// TIA Portal V17 export
// export: Created 2023-04-07T09:30:35.0113751Z, ExportSetting WithDefaults, DisplayName Totally Integrated Automation Portal, DisplayVersion V17 Update 4, DisplayName TIA Portal Openness, DisplayVersion V17 Update 4, DisplayName TIA Portal Version Control Interface, DisplayVersion V17, DisplayName STEP 7 Professional, DisplayVersion V17 Update 4, DisplayName STEP 7 Safety, DisplayVersion V17, DisplayName WinCC Professional, DisplayVersion V17 Update 4
TYPE "W_PE"
// stored: IsFailsafeCompliant false
   STRUCT
      iUserPswIns : Int;   // To check / 40005
      iModePctrlCmd : Int := 0;   // Register 40861 / 40551
      iModeQctrlCmd : Int := 0;   // Register 40862 / 40552
      rPacRef : Real := 0.0;   // Register 40863 / 40553
      rQacRef : Real := 0.0;   // Register 40864 / 40558
      xStartCmd : Bool;   // Register 40040
      xGeneral_SelectorEnable : Bool;   // Register 40039
      xDC_SelectorEnable : Bool;   // Register 40397
      xDC_VirtualSelector : Bool;   // Register 40398
      xAC_SelectorEnable : Bool;   // Register 40399
      xAC_VirtualSelector : Bool;   // Register 40400
      xStopCmd : Bool;   // Register 40041
      xClearFltCmd : Bool;   // To check
      xEmeStopCmd : Bool;   // Register 43039
      xEnableCmd : Bool;   // To check
      wBankDcEnbCmd : Word;   // To check
      iWatchDog : Int;   // To check
      xMVskid_comm : Bool;   // Register 41880 - 0 = communications enabled
      uiMVskid_CB : UInt;
   END_STRUCT;
END_TYPE
